// TwinCAT 3 PLC project MC
// ProgramVersion: 3.1.4022.4
// libraries:
//   Tc2_MC2, * (Beckhoff Automation GmbH)
//   Tc2_Standard, * (Beckhoff Automation GmbH)
//   Tc2_System, * (Beckhoff Automation GmbH)
//   Tc3_Module, * (Beckhoff Automation GmbH)
// project tree:
//   / GlobalTextList.TcGTLO, PlcTask.TcTTO, 视图管理器.TcVMO (not stored)
//   POUs/ LED.TcPOU, MAIN.TcPOU
//   VISUs/ HMI.TcVIS
// real-time tasks:
//   TASK PlcTask: cycle T#9ms, priority 19, ADS port 350
//   TASK Task 6: cycle T#10ms, priority 10, ADS port 351
// motion (NC):
//   TASK NC-Task 1 SAF: cycle T#2ms, priority 4, ADS port 501
//   TASK NC-Task 1 SVB: cycle T#10ms, priority 8, ADS port 511
//   AXIS Axis 6 (id 1)
//     General: UnitName=Degree
//     Dynamic: AccelerationMaximum=300, DecelerationMaximum=300, Acceleration=240, Deceleration=240, Jerk=400
//     Velo: RefSearch=20, RefSync=20, SlowManual=10, FastManual=20, Maximum=360
//     OtherSettings: AllowMotionCmdToSlave=true, PulseDistancePos=2, PulseDistanceNeg=2
//     encoder EncType=19
//       EncPara: ScaleFactorNumerator=36000, ScaleFactorDenominator=22648832, MaxCount=#xffffffff
//     drive DrvType=16
//       DrvPara: MaxCount=#xffffffff, DriveControlDWord=#x00020000
//         Analog: VeloReferenz=240, ScaleFactorActTorque=0.1
//         TimeComp: TaskDelayCycles=1
//     controller CtrType=1
//       CtrPara: PriorControlFactor=1
//         Observer: BandWidth=20
// I/O:
//   DEVICE Device 2 (EtherCAT), AmsNetId 192.168.1.116.3.1
//     Term 1 (EK1100) [EK1100 EtherCAT Coupler (2A E-Bus)]
//       Term 2 (EK1122) [EK1122 2 port EtherCAT junction]
//       Term 3 (EK1122) [EK1122 2 port EtherCAT junction]
//         Term 4 (EK1100) [EK1100 EtherCAT Coupler (2A E-Bus)]
//           Term 5 (EL2004) [EL2004 4Ch. Dig. Output 24V, 0.5A]
//           Term 6 (EL1008) [EL1008 8Ch. Dig. Input 24V, 3ms]
//           Term 7 (EL3162) [EL3162 2Ch. Ana. Input 0-10V]
//           Term 8 (EL6751) [EL6751 CANopen Master]
//           Term 14 (EL9011) [EL9011 End Terminal]
//         Term 9 (EK1100) [EK1100 EtherCAT Coupler (2A E-Bus)]
//           Term 10 (EL2004) [EL2004 4Ch. Dig. Output 24V, 0.5A]
//           Term 11 (EL1008) [EL1008 8Ch. Dig. Input 24V, 3ms]
//           Term 15 (EL9011) [EL9011 End Terminal]
//         Drive 12 (Elmo Drive) [Gold EtherCAT GCON Drive Rev:0x00010420]
//     Box 13 (M8126) [M8126]
//   DEVICE Device 1 (EL6751) (disabled), AmsNetId 192.168.1.116.2.1
// variable links:
//   Device 2 (EtherCAT) <-> MC_Cpp/MC_Cpp_Obj1 (Axis6)
//     Term 1 (EK1100)/Term 3 (EK1122)/Term 4 (EK1100)/Term 5 (EL2004)/Channel 1/Output <-> Outputs/led1
//   NC-Task 1 SAF/Axes/Axis 6 <-> Device 2 (EtherCAT)/Term 1 (EK1100)/Term 3 (EK1122)/Drive 12 (Elmo Drive)
//     Drive/Inputs/In/nDcOutputTime <-> InfoData/DcOutputShift
//     Drive/Inputs/In/nState1 <-> Inputs/Status word
//     Drive/Inputs/In/nState2 <-> Inputs/Status word @bit 8
//     Drive/Inputs/In/nState4 @bit 1 <-> WcState/InputToggle
//     Drive/Inputs/In/nState4 <-> WcState/WcState
//     Drive/Outputs/Out/nCtrl1 <-> Outputs/Control word
//     Drive/Outputs/Out/nCtrl2 <-> Outputs/Control word @bit 8
//     Drive/Outputs/Out/nDataOut1 <-> Outputs/Target Position
//     Enc/Inputs/In/nDataIn1 <-> Inputs/Position actual value
//     Enc/Inputs/In/nDcInputTime <-> InfoData/DcInputShift
//     Enc/Inputs/In/nState4 @bit 1 <-> WcState/InputToggle
//     Enc/Inputs/In/nState4 <-> WcState/WcState
//   MC/MC Instance <-> Device 2 (EtherCAT)/Term 1 (EK1100)/Term 3 (EK1122)/Term 4 (EK1100)/Term 6 (EL1008)
//     PlcTask Inputs/LED.SWITCH1 <-> Channel 1/Input
//   MC/MC Instance <-> NC-Task 1 SAF/Axes/Axis 6
//     PlcTask Inputs/MAIN.axis6.NcToPlc <-> Outputs/ToPlc
//     PlcTask Outputs/MAIN.axis6.PlcToNc <-> Inputs/FromPlc

CONFIGURATION MC
    RESOURCE PLC ON TwinCAT3
        TASK PlcTask(INTERVAL := T#9ms, PRIORITY := 19);
        PROGRAM MAIN WITH PlcTask : MAIN;
        PROGRAM LED WITH PlcTask : LED;
    END_RESOURCE
END_CONFIGURATION

// ---- POUs/MAIN.TcPOU
PROGRAM MAIN
VAR
	axis6: AXIS_REF;
	Power: MC_Power;

	power_do: BOOL;

	move_r: MC_MoveRelative;
	move_do: BOOL;
	set_position:MC_SetPosition;
	set_do: BOOL;
	reset:MC_Reset;
	reset_do: BOOL;
END_VAR

Power(
	Axis:= axis6, 
	Enable:= power_do, 
	Enable_Positive:= TRUE, 
	Enable_Negative:= TRUE, 
	Override:= , 
	BufferMode:= , 
	Options:= , 
	Status=> , 
	Busy=> , 
	Active=> , 
	Error=> , 
	ErrorID=> );

move_r(
	Axis:= axis6, 
	Execute:= move_do, 
	Distance:=360, 
	Velocity:=60 , 
	Acceleration:= 240, 
	Deceleration:= 240, 
	Jerk:= , 
	BufferMode:= , 
	Options:= , 
	Done=> , 
	Busy=> , 
	Active=> , 
	CommandAborted=> , 
	Error=> , 
	ErrorID=> );
set_position(
	Axis:= axis6, 
	Execute:= set_do, 
	Position:= 0, 
	Mode:= , 
	Options:= , 
	Done=> , 
	Busy=> , 
	Error=> , 
	ErrorID=> );
reset(
	Axis:=axis6 , 
	Execute:= reset_do, 
	Done=> , 
	Busy=> , 
	Error=> , 
	ErrorID=> );

END_PROGRAM

// ---- POUs/LED.TcPOU
PROGRAM LED
VAR
	
	LED1 AT%Q*: BOOL;
	SWITCH1 AT%I*: BOOL;
END_VAR

IF SWITCH1=1 THEN
	LED1:=1;
ELSE
	LED1:=0;
END_IF

END_PROGRAM

// ---- GlobalTextList.TcGTLO
TEXTLIST GlobalTextList
  699 = 'Axis6:%.2f'
  446 = 'Jog'
  564 = 'moveRelative'
  120 = 'Power'
  936 = 'reset'
  499 = 'setposition'
END_TEXTLIST

// ---- VISUs/HMI.TcVIS
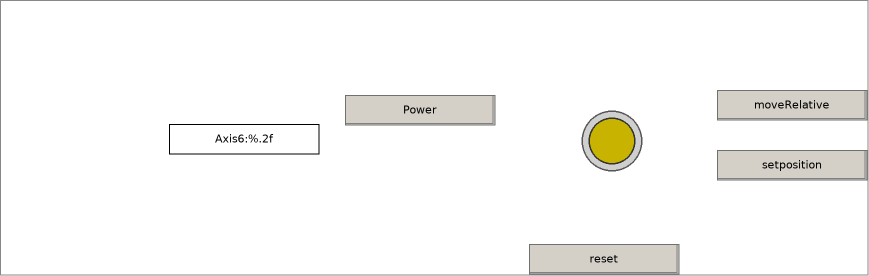
VISUALIZATION HMI  // 869x276
    Rectangle (169,124 150x30), "Axis6:%.2f", text variable: MAIN.axis6.NcToPlc.ActPos
    Button (345,95 150x30), "Power"
        toggle MAIN.power_do
    Lamp1 (577,106 70x70), variable: MAIN.axis6.NcToPlc.StateDWord.20, style: Lamp-Lamp1-Yellow
    Button (717,90 150x30), "moveRelative"
        tap MAIN.move_do
    Button (717,150 150x30), "setposition"
        tap MAIN.set_do
    Button (529,244 150x30), "reset"
        tap MAIN.reset_do
END_VISUALIZATION
